# B&R Automation Studio project AS (part 4)

#### Action_Set_Active_Rec.st
```iecst
ACTION Action_Set_Active_Rec:

	gRecipe_CSV_UIConnect.Recipe.List.SelectedIndex := 0;

	FOR ii_recipes := 0 TO MAX_IDX_TOTAL_RECIPES BY 1 DO
		IF (brsstrcmp(ADR(gRecipe_CSV_UIConnect.Recipe.List.Names[gRecipe_CSV_UIConnect.Recipe.List.SelectedIndex]), ADR(gRecipeName)) = 0) THEN
			EXIT;
		ELSE
			gRecipe_CSV_UIConnect.Recipe.List.StepDown := 1;
			Recipe_CSV_UI();
		END_IF;
	END_FOR;

END_ACTION
```

Listed in the project but not available here: Logical/Alarms.typ, Logical/Libraries/sscanf2/sscanf2.h, Logical/UserLibraries/jgLibs/VA_Setup/va_setup.c, Logical/UserLibraries/jgLibs/VA_Setup/VA_Setup.fun, Logical/UserLibraries/jgLibs/jgUtils/Types.typ, Logical/UserLibraries/jgLibs/jgUtils/HW_modules.typ, Logical/UserLibraries/jgLibs/jgUtils/Constants.var, Logical/UserLibraries/jgLibs/jgUtils/jgUtils.fun, Logical/UserLibraries/wbrServices/Doc, Logical/UserLibraries/wbrServices/wbrServices_C_Includes, Logical/UserLibraries/wbrServices/wbrMemSvc/wbrMemSvc.typ, Logical/UserLibraries/wbrServices/wbrMemSvc/wbrMemSvc.fun, Logical/UserLibraries/wbrServices/wbrLogSvc/wbrLogSvc.typ, Logical/UserLibraries/wbrServices/wbrLogSvc/wbrLogSvc.var, Logical/UserLibraries/wbrServices/wbrLogSvc/wbrLogSvc.fun, Logical/UserLibraries/wbrServices/wbrPingSvc/wbrPingSvc.typ, Logical/UserLibraries/wbrServices/wbrPingSvc/wbrPingSvc.fun, Logical/UserLibraries/wbrServices/wbrPingSvc/wbrPingSvc.c, Logical/UserLibraries/wbrServices/wbrSvcUtilities/wbrBitUtil/wbrBitUtil.typ, Logical/UserLibraries/wbrServices/wbrSvcUtilities/wbrBitUtil/wbrBitUtil.fun, Logical/UserLibraries/wbrServices/InitSP/appConfig.typ, Logical/UserLibraries/wbrServices/Cyclic/wbrService, Logical/Application_Logic/pkgDispense/Dispense/Main.st, Logical/Application_Logic/pkgDispense/Dispense/Types.typ, Logical/Application_Logic/pkgDispense/Dispense/Variables.var, Logical/Application_Logic/pkgDispense/Dispense/libDisp.fun, Logical/Application_Logic/pkgDispense/Dispense/HernonDispValve.st, Logical/Application_Logic/pkgDispense/HMITableTexts, Logical/Application_Logic/pkgDispense/libDisp/Disp_StateMachine_States.typ, Logical/Application_Logic/pkgDispense/libDisp/Disp_Belt_Types.typ, Logical/Application_Logic/pkgDispense/libDisp/Constants.var, Logical/Application_Logic/pkgDispense/libDisp/libDisp.fun, Logical/Application_Logic/pkgInspect/Inspect/Types.typ, Logical/Application_Logic/pkgInspect/libInsp/Insp_IO.typ, Logical/Application_Logic/pkgInspect/libInsp/Constants.var, Logical/Application_Logic/pkgInspect/libInsp/libInsp.fun, Logical/paiComponents/bglib/bgXmlRpcParser.h, Logical/paiComponents/bglib/_X_bgftpclient.c, Logical/paiComponents/bglib/bgBitUtilities.h, Logical/paiComponents/bglib/bgBitUtilities.c, Logical/paiComponents/bglib/bgBufMemAlloc.h, Logical/paiComponents/bglib/bgBufMemAlloc.c, Logical/paiComponents/bglib/bgDataStructures.h, Logical/paiComponents/bglib/bgDataStructures.c, Logical/paiComponents/bglib/bgdebugV2.h, Logical/paiComponents/bglib/bgfsig.h, Logical/paiComponents/bglib/bgfsig.c, Logical/paiComponents/bglib/bgftpclient.h, Logical/paiComponents/bglib/bgftpclient.c, Logical/paiComponents/bglib/bgftpclient_lib.c, Logical/paiComponents/bglib/bgHttpAppWeb.h, Logical/paiComponents/bglib/bgHttpAppWeb.c, Logical/paiComponents/bglib/bgHttpAppXmlRpc.h, Logical/paiComponents/bglib/bgHttpAppXmlRpc.c, Logical/paiComponents/bglib/bgHttpProtocol.h, Logical/paiComponents/bglib/bgHttpProtocol.c, Logical/paiComponents/bglib/bglibversion.h, Logical/paiComponents/bglib/bglib-1.c, Logical/paiComponents/bglib/bglib.c, Logical/paiComponents/bglib/bgPVLogger2.c, Logical/paiComponents/bglib/bgPVLogger3.c, Logical/paiComponents/bglib/bgPVLogger.c, Logical/paiComponents/bglib/bgringbuffer.h, Logical/paiComponents/bglib/bgringbuffer.c, Logical/paiComponents/bglib/bgSecMD5Signature.h, Logical/paiComponents/bglib/bgSecMD5Signature.c, Logical/paiComponents/bglib/bgsscanf.h, Logical/paiComponents/bglib/bgsscanf.c, Logical/paiComponents/bglib/bgstatemachine.h, Logical/paiComponents/bglib/bgstatemachine.c, Logical/paiComponents/bglib/bgstring.h, Logical/paiComponents/bglib/bgstring.c, Logical/paiComponents/bglib/bgstringTest.c, Logical/paiComponents/bglib/bgTcpSocketClientServer.h, Logical/paiComponents/bglib/bgTcpSocketClient.c, Logical/paiComponents/bglib/bgTcpSocketServer.c, Logical/paiComponents/bglib/bgTimer.h, Logical/paiComponents/bglib/bgTimer1ms.h, Logical/paiComponents/bglib/bgTimer1ms.c, Logical/paiComponents/bglib/bgTimer.c, Logical/paiComponents/bglib/bgXmlRpcParser.c, Logical/paiComponents/bglib/bgPVSerializeJSON.h, Logical/paiComponents/bglib/bgPVSerialize.h, Logical/paiComponents/bglib/bgPVSerialize.c, Logical/paiComponents/bglib/bgTelnetSrvr-astcpV2.c, Logical/paiComponents/bglib/bgTelnetSrvr-astcpV2.h, Logical/paiComponents/Libraries/bgringbuf/bgringbuffer.h, Logical/paiComponents/Libraries/bgringbuf/bgringbuffer.c, Logical/paiComponents/paiFileService/paiPVSerDesMgr.typ, Logical/paiComponents/paiFileService/paiFileService.typ, Logical/paiComponents/paiFileService/paiFileService.var, Logical/paiComponents/paiFileService/paiFS/paiFile.c, Logical/paiComponents/paiFileService/paiFS/paiDevDirConfigure.c, Logical/paiComponents/bglib/bgstring.c, Logical/paiComponents/paiFileService/paiFSUnitTest/paiFSUnitTest.c, Logical/paiComponents/paiFileService/paiPVSerDesMgr.h, Logical/paiComponents/paiFileService/paiFSInterface.h, Logical/paiComponents/paiFileService/paiFSInterface.c, Logical/paiComponents/paiHmi/paiHmiTemplate.typ, Logical/paiComponents/paiHmi/paiARSystem.typ, Logical/paiComponents/paiHmi/paiHmiDialog.typ, Logical/paiComponents/paiHmi/paiHmiMsgRunning.typ, Logical/paiComponents/paiHmi/paiHmiMsgScroll.typ, Logical/paiComponents/paiHmi/paiHmiAlert.typ, Logical/paiComponents/paiHmi/paiHmiSystemNetworking.typ, Logical/paiComponents/paiHmi/paiHmiSystemDateTime.typ, Logical/paiComponents/paiHmi/paiHmiCmd.typ, Logical/paiComponents/paiHmi/paiHmiStatus.typ, Logical/paiComponents/paiHmi/paiHmiDialog.h, Logical/paiComponents/paiHmi/paiHmiDialog.c, Logical/paiComponents/paiHmi/paiHmiPageChange.h, Logical/paiComponents/paiHmi/paiHmiPageChange.c, Logical/paiComponents/paiHmi/paiHmiAlert.c, Logical/paiComponents/paiHmi/paiHmiSystemNetworking.h, Logical/paiComponents/paiHmi/paiHmiSystemNetworking.c, Logical/paiComponents/paiHmi/paiHmiSystemDateTime.h, Logical/paiComponents/paiHmi/paiHmiTableViewProducts.c, Logical/paiComponents/paiHmi/paiHmiTableViewPersons.c, Logical/paiComponents/paiHmi/paiHmiParamList.c, Logical/paiComponents/paiHmi/paiHmiLFMenuTabsPages.h, Logical/paiComponents/paiHmi/paiHmiLFMenuTabsPages.c, Logical/paiComponents/paiHmi/paiHmiMsgScrolling.h, Logical/paiComponents/paiHmi/paiHmiMsgScrolling.c, Logical/paiComponents/paiHmi/paiHmiDropdownMenuRT.h, Logical/paiComponents/paiHmi/paiHmiDropdownMenuRT.c, Logical/paiComponents/paiPing/paiPingService, Logical/paiComponents/paiTemplate/paiHMI/paiHmi/paiHmi.c, Logical/paiComponents/bglib/bgstring.c, Logical/paiComponents/bglib/bgBitUtilities.c, Logical/paiComponents/paiHmi/paiHmiLFMenuTabsPages.c, Logical/paiComponents/paiHmi/paiHmiAlert.c, Logical/paiComponents/paiHmi/paiHmiDialog.c, Logical/paiComponents/paiHmi/paiHmiMsgScrolling.c, Logical/paiComponents/paiHmi/paiHmiDropdownMenuRT.c, Logical/paiComponents/paiHmi/paiHmiSystemNetworking.c, Logical/paiComponents/paiUDP/udpApp.typ, Logical/paiComponents/paiUDP/udpApp.var, Logical/paiComponents/paiUDP/paiUDPService, Logical/paiComponents/paiUDP/udpApp, Logical/paiComponents/paiUser/paiUser/paiUser.c, Logical/pkgSafety/SafeINIT/Main.st, Logical/pkgSafety/SafeINIT/Types.typ, Logical/pkgSafety/SafeINIT/Variables.var, Logical/pkgSafety/SafeINIT/Action_Init_RCTRL_Cmd.st, Logical/HMI/HMI_Page_Enum.typ, Logical/pkgRecCfg/Recipe_Handling/Cyclic.st, Logical/pkgRecCfg/Recipe_Handling/Exit.st, Logical/pkgRecCfg/Recipe_Handling/Types.typ, Logical/pkgRecCfg/Recipe_Handling/Variables.var, Logical/pkgRecCfg/Recipe_Handling/Action_Set_Active_Rec.st, Logical/pkgRecCfg/Recipe_Handling/LocalFunctions.fun, Logical/pkgAlert/ComLogger, Logical/pkgAccess/UserX, Logical/pkgData/DataTask/Main.st, Logical/pkgData/DataTask/Types.typ, Logical/pkgData/DataTask/Variables.var, Logical/pkgData/File_Handling/Cyclic.st, Logical/pkgData/File_Handling/Exit.st, Logical/pkgData/File_Handling/Types.typ, Logical/pkgData/File_Handling/Variables.var, Logical/pkgPVListView/TableIndex_Enum.typ, Logical/pkgPVListView/pvListView_Global_Var.var, Logical/pkgPVListView/paiPVTable/HMIparamList.typ, Logical/pkgPVListView/paiPVTable/Constants.var, Logical/pkgPVListView/paiPVTable/paiPVTable.fun, Logical/pkgPVListView/paiPVTable/hmiParamList.h, Logical/pkgPVListView/paiPVTable/hmiParamList.c, Logical/pkgPVListView/paiPVTable/bgstring.c, Logical/pkgPVListView/paiPVTable/bgstring.h, Logical/pkgPVListView/paiPVTable/bgsprintf.c, Logical/pkgPVListView/paiPVTable/bgsprintf.h, Logical/pkgPVListView/paiPVTable/hmiTableFBK_typ.c, Logical/pkgPVListView/paiPVTable/ActivateHMITable.c, Logical/pkgOEE, Logical/GmcIpConfig/gmciplbr, Logical/GmcIpConfig/gmcipesm, Logical/GmcIpConfig/gmcipmx, Logical/Application/Dispense/Texts/Params/Recipe, Logical/Application/Dispense/Texts/Params/Config
